SUBAPPLICATION SubApp_PC_B (* Geraet B (Station 12, 192.168.1.12): empfaengt Hoch/Runter-Zustand per OPC-UA (AX_SUBSCRIBE_1, lokal ueberwacht), fuehrt beide direkt per Adapter-Verbindung in ILOCK_SWITCH_PROTECT_AX (Last-Wins mit Schutzzeit) zusammen und schaltet Output_Q7/Output_Q8 - 'SUB style': das FB-Netz steckt direkt in diesem Composite, da diese Kombination (2x Subscribe + Interlock + Schutzzeit-Timer + 2x Ausgang) exercise-spezifisch ist. AX_SUBSCRIBE_1.OUT ist bereits vom Adaptertyp 'AX' - demselben Typ, den ILOCK_SWITCH_PROTECT_AX.UP_IN/.DOWN_IN als Socket erwarten - daher keine Zwischen-Logik noetig (Vorbild fuer die ILOCK-Verdrahtung selbst: test_AX/Uebungen/Uebung_202_AX.SUB) *)
  (* Standard: 61499-2; Description: Copyright (c) 2026 Meisterschulen am Ostbahnhof This program and the accompanying materials are made available under the terms of the Eclipse Public License 2.0 which is available at https://www.eclipse.org/legal/epl-2.0/ SPDX-License-Identifier: EPL-2.0 *)
  (* Version 1.0, 2026-09-05, Franz Höpfinger, Meisterschulen am Ostbahnhof, initial API and implementation and/or initial documentation *)
  PACKAGE subapp::Training_10_OPC_UA_RES;
  IMPORT VV::const::OPC_UA::myOpcUaAddresses::SW1_UP_LOCAL_READ;
  IMPORT VV::const::OPC_UA::myOpcUaAddresses::SW1_DOWN_LOCAL_READ;
  IMPORT logiBUS::io::DQ::logiBUS_DO::Output_Q7;
  IMPORT logiBUS::io::DQ::logiBUS_DO::Output_Q8;
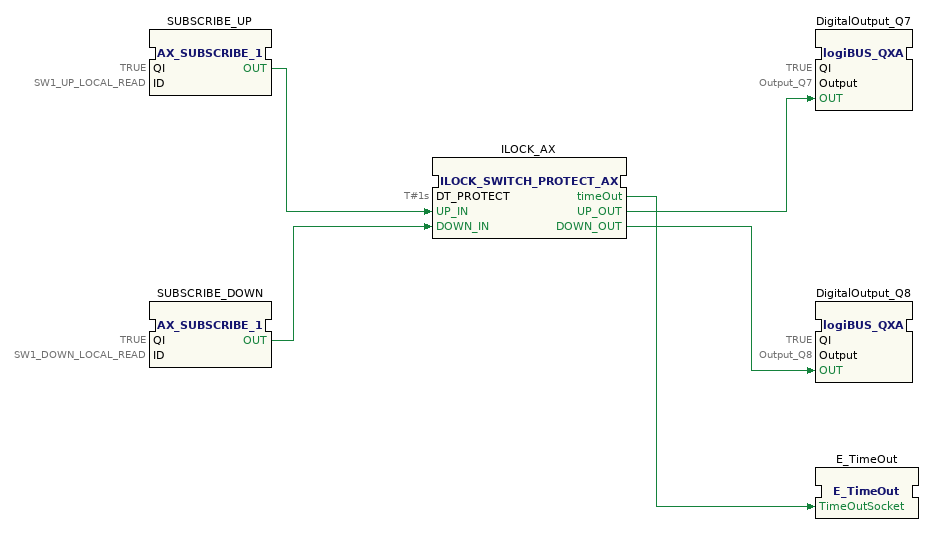
  FBS
    SUBSCRIBE_UP : adapter::net::AX_SUBSCRIBE_1(QI := TRUE, ID := SW1_UP_LOCAL_READ);
    SUBSCRIBE_DOWN : adapter::net::AX_SUBSCRIBE_1(QI := TRUE, ID := SW1_DOWN_LOCAL_READ);
    ILOCK_AX : logiBUS::signalprocessing::interlock::ILOCK_SWITCH_PROTECT_AX(DT_PROTECT := T#1s);
    E_TimeOut : iec61499::events::E_TimeOut;
    DigitalOutput_Q7 : logiBUS::io::DQ::logiBUS_QXA(QI := TRUE, Output := Output_Q7);
    DigitalOutput_Q8 : logiBUS::io::DQ::logiBUS_QXA(QI := TRUE, Output := Output_Q8);
  END_FBS
  ADAPTER_CONNECTIONS
    SUBSCRIBE_UP.OUT TO ILOCK_AX.UP_IN;
    SUBSCRIBE_DOWN.OUT TO ILOCK_AX.DOWN_IN;
    ILOCK_AX.timeOut TO E_TimeOut.TimeOutSocket;
    ILOCK_AX.UP_OUT TO DigitalOutput_Q7.OUT;
    ILOCK_AX.DOWN_OUT TO DigitalOutput_Q8.OUT;
  END_CONNECTIONS
END_SUBAPPLICATION
